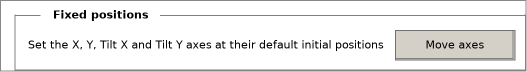
VISUALIZATION VISU_M2Fixed  // 527x72
VAR_IN_OUT
	ref : M2;
    widget : M2Widget;
END_VAR
    Polyline (160,15) (525,15) (525,70) (15,70) (15,15) (40,15)
    Label (25,35 380x20), "Set the X, Y, Tilt X and Tilt Y axes at their default initial positions"
    Label (50,5 115x20), "Fixed positions"
    Button (395,30 120x30), "Move axes", input disabled if: ref.processes.verifyFixedPositions.statuses.enabledStatus.disabled
        OnMouseClick: execute { ref.processes.verifyFixedPositions.do_request := TRUE; }
END_VISUALIZATION

(* stored: Version 1.1.0.1, ProductVersion 3.1.4018.5
   Visu VISU_M2Fixed: Id {368c2d97-7e92-46d0-8f5c-9b4b58a67881} *)
